INTERFACE I_Base EXTENDS __SYSTEM.IQueryInterface

END_INTERFACE

(* stored: Version 1.1.0.1
   Itf I_Base: Id {0febec6b-070a-4fab-983e-e57bba388fd2} *)
